% RSLogix 500 project PROJECT10.RSS, saved by version 8.30.00.16 %
PROJECT "FINAL"    % processor: Bul.1763 MicroLogix 1100 Series B %

PROGRAM FILES
  LAD 2 "MAIN"  6 rungs
  LAD 3 "IO"  10 rungs
  LAD 4 "HOA CTRL"  7 rungs
  LAD 5 "ALARMS"  12 rungs
  LAD 6 "AUTO RUN"  5 rungs

DATA FILES
  O0 OUTPUT  4 elements
  I1 INPUT  6 elements
  S2 STATUS  66 elements
  B3 BINARY  2 elements
  T4 TIMER  5 elements
  C5 COUNTER  1 elements
  R6 CONTROL  1 elements
  N7 INTEGER  4 elements
  F8 FLOAT  1 elements

LADDER 2 "MAIN"
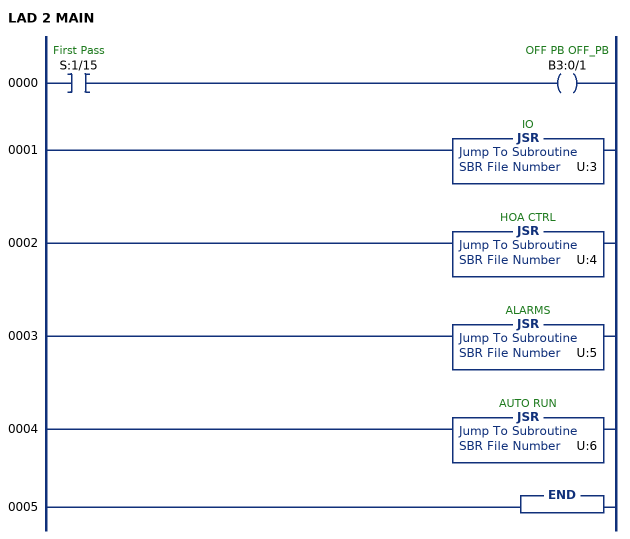
% Rung: 0 %
SOR XIC S:1/15 OTE B3:0/1 EOR
%   S:1/15  "First Pass" %
%   B3:0/1  OFF_PB  "OFF PB" %
% Rung: 1 %
SOR JSR U:3 EOR
%   U:3  "IO" %
% Rung: 2 %
SOR JSR U:4 EOR
%   U:4  "HOA CTRL" %
% Rung: 3 %
SOR JSR U:5 EOR
%   U:5  "ALARMS" %
% Rung: 4 %
SOR JSR U:6 EOR
%   U:6  "AUTO RUN" %
% Rung: 5 %
SOR END EOR

LADDER 3 "IO"
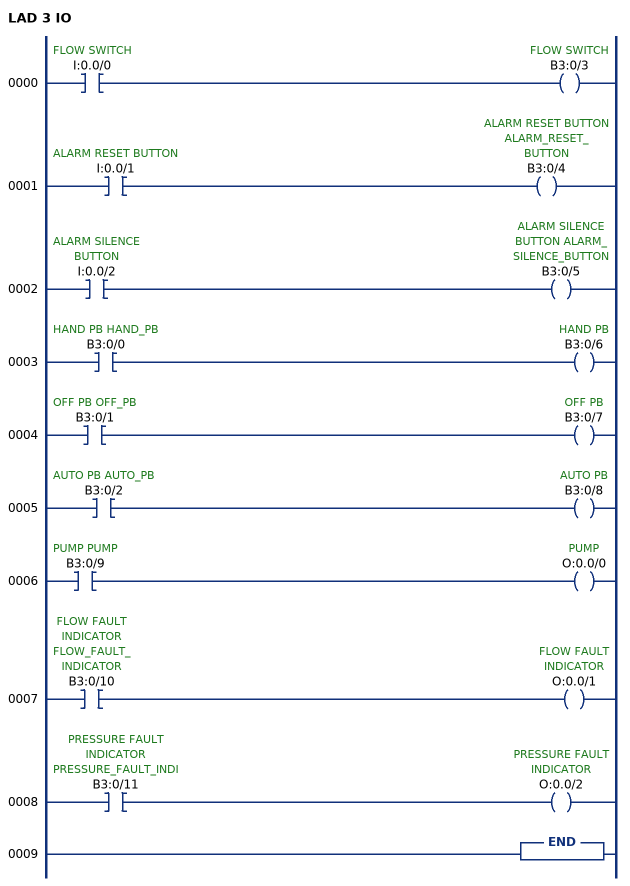
% Rung: 0 %
SOR XIC I:0.0/0 OTE B3:0/3 EOR
%   I:0.0/0  "FLOW SWITCH" %
%   B3:0/3  "FLOW SWITCH" %
% Rung: 1 %
SOR XIC I:0.0/1 OTE B3:0/4 EOR
%   I:0.0/1  "ALARM RESET BUTTON" %
%   B3:0/4  ALARM_RESET_BUTTON  "ALARM RESET BUTTON" %
% Rung: 2 %
SOR XIC I:0.0/2 OTE B3:0/5 EOR
%   I:0.0/2  "ALARM SILENCE BUTTON" %
%   B3:0/5  ALARM_SILENCE_BUTTON  "ALARM SILENCE BUTTON" %
% Rung: 3 %
SOR XIC B3:0/0 OTE B3:0/6 EOR
%   B3:0/0  HAND_PB  "HAND PB" %
%   B3:0/6  "HAND PB" %
% Rung: 4 %
SOR XIC B3:0/1 OTE B3:0/7 EOR
%   B3:0/1  OFF_PB  "OFF PB" %
%   B3:0/7  "OFF PB" %
% Rung: 5 %
SOR XIC B3:0/2 OTE B3:0/8 EOR
%   B3:0/2  AUTO_PB  "AUTO PB" %
%   B3:0/8  "AUTO PB" %
% Rung: 6 %
SOR XIC B3:0/9 OTE O:0.0/0 EOR
%   B3:0/9  PUMP  "PUMP" %
%   O:0.0/0  "PUMP" %
% Rung: 7 %
SOR XIC B3:0/10 OTE O:0.0/1 EOR
%   B3:0/10  FLOW_FAULT_INDICATOR  "FLOW FAULT INDICATOR" %
%   O:0.0/1  "FLOW FAULT INDICATOR" %
% Rung: 8 %
SOR XIC B3:0/11 OTE O:0.0/2 EOR
%   B3:0/11  PRESSURE_FAULT_INDI  "PRESSURE FAULT INDICATOR" %
%   O:0.0/2  "PRESSURE FAULT INDICATOR" %
% Rung: 9 %
SOR END EOR

LADDER 4 "HOA CTRL"
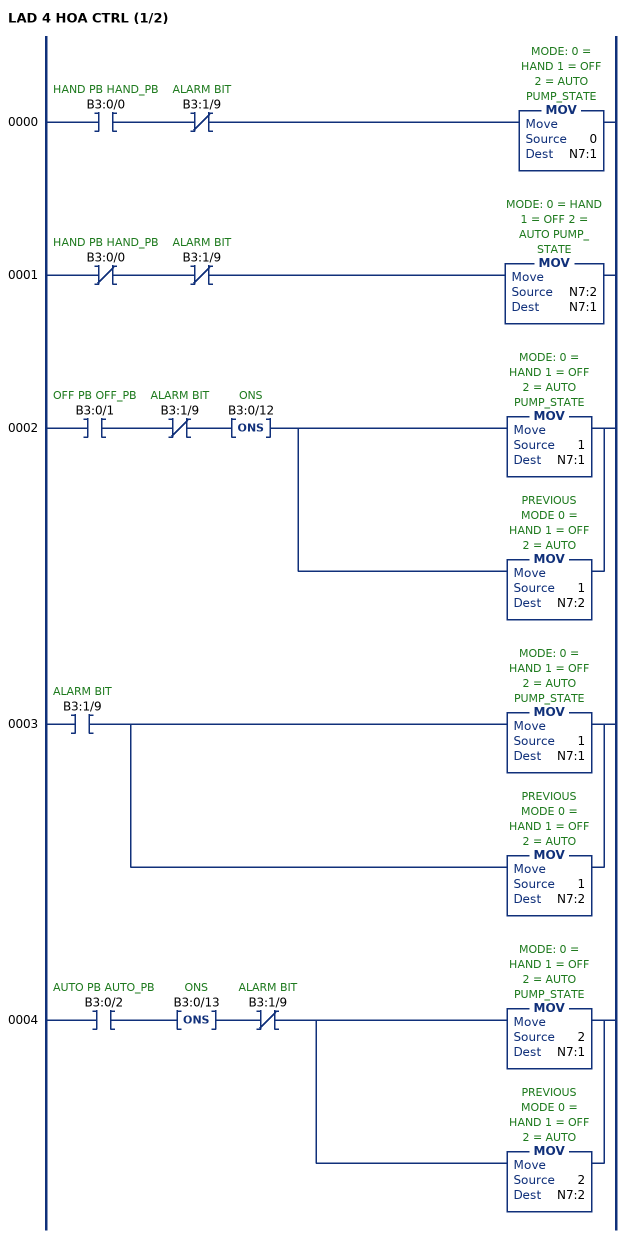
% Rung: 0 %
SOR XIC B3:0/0 XIO B3:1/9 MOV 0 N7:1 EOR
%   B3:0/0  HAND_PB  "HAND PB" %
%   B3:1/9  "ALARM BIT" %
%   N7:1  PUMP_STATE  "MODE: 0 = HAND 1 = OFF 2 = AUTO" %
% Rung: 1 %
SOR XIO B3:0/0 XIO B3:1/9 MOV N7:2 N7:1 EOR
%   B3:0/0  HAND_PB  "HAND PB" %
%   B3:1/9  "ALARM BIT" %
%   N7:2  "PREVIOUS MODE 0 = HAND 1 = OFF 2 = AUTO" %
%   N7:1  PUMP_STATE  "MODE: 0 = HAND 1 = OFF 2 = AUTO" %
% Rung: 2 %
SOR XIC B3:0/1 XIO B3:1/9 ONS B3:0/12 BST MOV 1 N7:1 NXB MOV 1 N7:2 BND EOR
%   B3:0/1  OFF_PB  "OFF PB" %
%   B3:1/9  "ALARM BIT" %
%   B3:0/12  "ONS" %
%   N7:1  PUMP_STATE  "MODE: 0 = HAND 1 = OFF 2 = AUTO" %
%   N7:2  "PREVIOUS MODE 0 = HAND 1 = OFF 2 = AUTO" %
% Rung: 3 %
SOR XIC B3:1/9 BST MOV 1 N7:1 NXB MOV 1 N7:2 BND EOR
%   B3:1/9  "ALARM BIT" %
%   N7:1  PUMP_STATE  "MODE: 0 = HAND 1 = OFF 2 = AUTO" %
%   N7:2  "PREVIOUS MODE 0 = HAND 1 = OFF 2 = AUTO" %
% Rung: 4 %
SOR XIC B3:0/2 ONS B3:0/13 XIO B3:1/9 BST MOV 2 N7:1 NXB MOV 2 N7:2 BND EOR
%   B3:0/2  AUTO_PB  "AUTO PB" %
%   B3:0/13  "ONS" %
%   B3:1/9  "ALARM BIT" %
%   N7:1  PUMP_STATE  "MODE: 0 = HAND 1 = OFF 2 = AUTO" %
%   N7:2  "PREVIOUS MODE 0 = HAND 1 = OFF 2 = AUTO" %

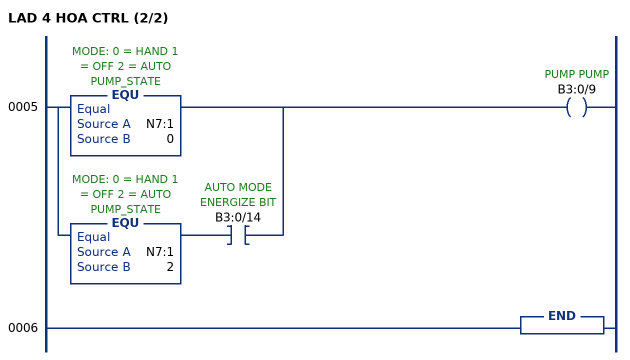
% Rung: 5 %
SOR BST EQU N7:1 0 NXB EQU N7:1 2 XIC B3:0/14 BND OTE B3:0/9 EOR
%   N7:1  PUMP_STATE  "MODE: 0 = HAND 1 = OFF 2 = AUTO" %
%   B3:0/14  "AUTO MODE ENERGIZE BIT" %
%   B3:0/9  PUMP  "PUMP" %
% Rung: 6 %
SOR END EOR

LADDER 5 "ALARMS"
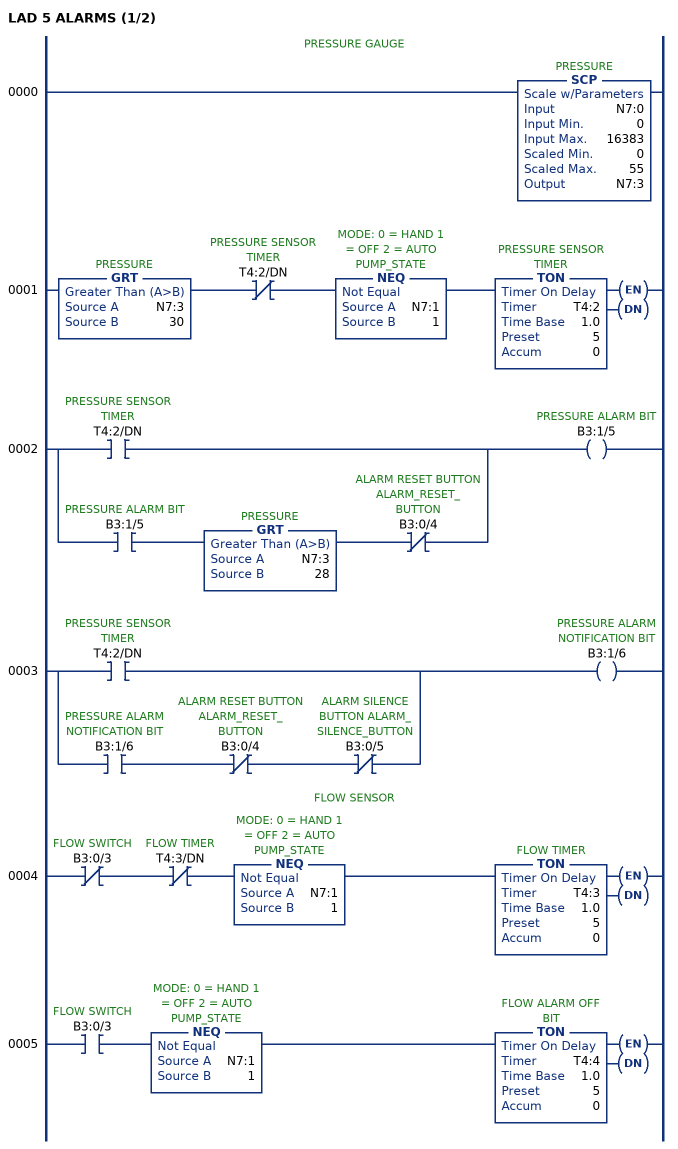
% Rung: 0 %
% PRESSURE GAUGE %
SOR SCP N7:0 0 16383 0 55 N7:3 EOR
%   N7:0  "PRESSURE SENSOR" %
%   N7:3  "PRESSURE" %
% Rung: 1 %
SOR GRT N7:3 30 XIO T4:2/DN NEQ N7:1 1 TON T4:2 1.0 5 0 EOR
%   N7:3  "PRESSURE" %
%   T4:2  "PRESSURE SENSOR TIMER" %
%   N7:1  PUMP_STATE  "MODE: 0 = HAND 1 = OFF 2 = AUTO" %
% Rung: 2 %
SOR BST XIC T4:2/DN NXB XIC B3:1/5 GRT N7:3 28 XIO B3:0/4 BND OTE B3:1/5 EOR
%   T4:2  "PRESSURE SENSOR TIMER" %
%   B3:1/5  "PRESSURE ALARM BIT" %
%   N7:3  "PRESSURE" %
%   B3:0/4  ALARM_RESET_BUTTON  "ALARM RESET BUTTON" %
% Rung: 3 %
SOR BST XIC T4:2/DN NXB XIC B3:1/6 XIO B3:0/4 XIO B3:0/5 BND OTE B3:1/6 EOR
%   T4:2  "PRESSURE SENSOR TIMER" %
%   B3:1/6  "PRESSURE ALARM NOTIFICATION BIT" %
%   B3:0/4  ALARM_RESET_BUTTON  "ALARM RESET BUTTON" %
%   B3:0/5  ALARM_SILENCE_BUTTON  "ALARM SILENCE BUTTON" %
% Rung: 4 %
% FLOW SENSOR %
SOR XIO B3:0/3 XIO T4:3/DN NEQ N7:1 1 TON T4:3 1.0 5 0 EOR
%   B3:0/3  "FLOW SWITCH" %
%   T4:3  "FLOW TIMER" %
%   N7:1  PUMP_STATE  "MODE: 0 = HAND 1 = OFF 2 = AUTO" %
% Rung: 5 %
SOR XIC B3:0/3 NEQ N7:1 1 TON T4:4 1.0 5 0 EOR
%   B3:0/3  "FLOW SWITCH" %
%   N7:1  PUMP_STATE  "MODE: 0 = HAND 1 = OFF 2 = AUTO" %
%   T4:4  "FLOW ALARM OFF BIT" %

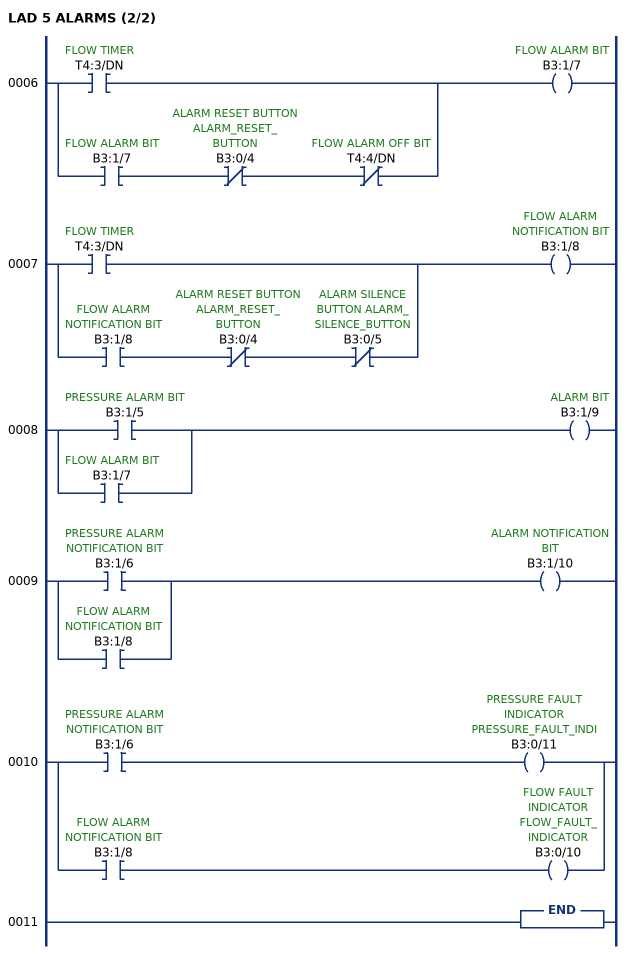
% Rung: 6 %
SOR BST XIC T4:3/DN NXB XIC B3:1/7 XIO B3:0/4 XIO T4:4/DN BND OTE B3:1/7 EOR
%   T4:3  "FLOW TIMER" %
%   B3:1/7  "FLOW ALARM BIT" %
%   B3:0/4  ALARM_RESET_BUTTON  "ALARM RESET BUTTON" %
%   T4:4  "FLOW ALARM OFF BIT" %
% Rung: 7 %
SOR BST XIC T4:3/DN NXB XIC B3:1/8 XIO B3:0/4 XIO B3:0/5 BND OTE B3:1/8 EOR
%   T4:3  "FLOW TIMER" %
%   B3:1/8  "FLOW ALARM NOTIFICATION BIT" %
%   B3:0/4  ALARM_RESET_BUTTON  "ALARM RESET BUTTON" %
%   B3:0/5  ALARM_SILENCE_BUTTON  "ALARM SILENCE BUTTON" %
% Rung: 8 %
SOR BST XIC B3:1/5 NXB XIC B3:1/7 BND OTE B3:1/9 EOR
%   B3:1/5  "PRESSURE ALARM BIT" %
%   B3:1/7  "FLOW ALARM BIT" %
%   B3:1/9  "ALARM BIT" %
% Rung: 9 %
SOR BST XIC B3:1/6 NXB XIC B3:1/8 BND OTE B3:1/10 EOR
%   B3:1/6  "PRESSURE ALARM NOTIFICATION BIT" %
%   B3:1/8  "FLOW ALARM NOTIFICATION BIT" %
%   B3:1/10  "ALARM NOTIFICATION BIT" %
% Rung: 10 %
SOR BST XIC B3:1/6 OTE B3:0/11 NXB XIC B3:1/8 OTE B3:0/10 BND EOR
%   B3:1/6  "PRESSURE ALARM NOTIFICATION BIT" %
%   B3:0/11  PRESSURE_FAULT_INDI  "PRESSURE FAULT INDICATOR" %
%   B3:1/8  "FLOW ALARM NOTIFICATION BIT" %
%   B3:0/10  FLOW_FAULT_INDICATOR  "FLOW FAULT INDICATOR" %
% Rung: 11 %
SOR END EOR

LADDER 6 "AUTO RUN"
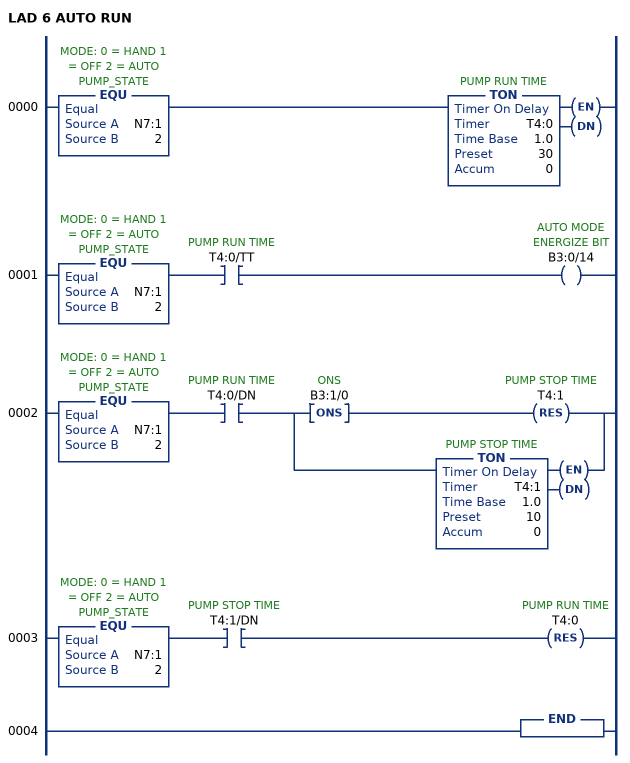
% Rung: 0 %
SOR EQU N7:1 2 TON T4:0 1.0 30 0 EOR
%   N7:1  PUMP_STATE  "MODE: 0 = HAND 1 = OFF 2 = AUTO" %
%   T4:0  "PUMP RUN TIME" %
% Rung: 1 %
SOR EQU N7:1 2 XIC T4:0/TT OTE B3:0/14 EOR
%   N7:1  PUMP_STATE  "MODE: 0 = HAND 1 = OFF 2 = AUTO" %
%   T4:0  "PUMP RUN TIME" %
%   B3:0/14  "AUTO MODE ENERGIZE BIT" %
% Rung: 2 %
SOR EQU N7:1 2 XIC T4:0/DN BST ONS B3:1/0 RES T4:1 NXB TON T4:1 1.0 10 0 BND EOR
%   N7:1  PUMP_STATE  "MODE: 0 = HAND 1 = OFF 2 = AUTO" %
%   T4:0  "PUMP RUN TIME" %
%   B3:1/0  "ONS" %
%   T4:1  "PUMP STOP TIME" %
% Rung: 3 %
SOR EQU N7:1 2 XIC T4:1/DN RES T4:0 EOR
%   N7:1  PUMP_STATE  "MODE: 0 = HAND 1 = OFF 2 = AUTO" %
%   T4:1  "PUMP STOP TIME" %
%   T4:0  "PUMP RUN TIME" %
% Rung: 4 %
SOR END EOR

OTHER DOCUMENTED ADDRESSES
  B3:0/15  "ALARM BIT"
  B3:1/1  "ONS"
  B3:1/3  "INITIAL COND."

DATA TABLE (non-zero values as saved)
DATA T4
% .PRE .ACC %
% T4:0 % 30 0
% T4:1 % 10 0
% T4:2 % 5 0
% T4:3 % 5 0
% T4:4 % 5 0
